FUNCTION_BLOCK SlaveAxisControl EXTENDS MasterAxisControl
VAR
	
	_PreviousAnglePosition		: LREAL;
	_PreviousLengthOfShaft		: LREAL;
	_PreviousWidthOfShaft		: LREAL;
	
	_xCoordPreviousRelative		: LREAL;
	_yCoordPreviousRelative		: LREAL;
	_xCoordPreviousGlobal		: LREAL;
	_yCoordPreviousGlobal		: LREAL;
	_xCoordGlobal				: LREAL;
	_yCoordGlobal				: LREAL;
	
	_SlaveOrderInChain			: LREAL;
	
END_VAR

METHOD CyclicUpdate : BOOL
VAR_INPUT
END_VAR
_Enable(Axis := _Axis);
_Reset(Axis := _Axis);
_ReadStatus(Axis := _Axis);
_MovePosAbs(Axis := _Axis);
_MovePosRel(Axis := _Axis);

_AnglePosition := _Axis.NcToPlc.ModuloActPos;

_xCoordRelative := _PreviousLengthOfShaft * COS(_PreviousAnglePosition * Pi / 180);
_yCoordRelative := _PreviousLengthOfShaft * SIN(_PreviousAnglePosition * Pi / 180);

_xCoordGlobal := _xCoordRelative + _xCoordPreviousGlobal;
_yCoordGlobal := _yCoordRelative + _yCoordPreviousGlobal;
END_METHOD

PROPERTY PreviousAnglePosition : LREAL
GET
PreviousAnglePosition := _PreviousAnglePosition;
END_GET
SET
_PreviousAnglePosition := PreviousAnglePosition;
END_SET
END_PROPERTY

PROPERTY PreviousLengthOfShaft : LREAL
GET
PreviousLengthOfShaft := _PreviousLengthOfShaft;
END_GET
SET
_PreviousLengthOfShaft := PreviousLengthOfShaft;
END_SET
END_PROPERTY

PROPERTY PreviousWidthOfShaft : LREAL
GET
PreviousWidthOfShaft := _PreviousWidthOfShaft;
END_GET
SET
_PreviousWidthOfShaft := PreviousWidthOfShaft;
END_SET
END_PROPERTY

PROPERTY PreviousXCoordGlobal : LREAL
GET
PreviousXCoordGlobal := _xCoordPreviousGlobal;
END_GET
SET
_xCoordPreviousGlobal := PreviousXCoordGlobal;
END_SET
END_PROPERTY

PROPERTY PreviousXCoordRelative : LREAL
GET
PreviousXCoordRelative := _xCoordPreviousRelative;
END_GET
SET
_xCoordPreviousRelative := PreviousXCoordRelative;
END_SET
END_PROPERTY

PROPERTY PreviousYCoordGlobal : LREAL
GET
PreviousYCoordGlobal := _yCoordPreviousGlobal;
END_GET
SET
_yCoordPreviousGlobal := PreviousYCoordGlobal;
END_SET
END_PROPERTY

PROPERTY PreviousYCoordRelative : LREAL
GET
PreviousYCoordRelative := _yCoordPreviousRelative;
END_GET
SET
_yCoordPreviousRelative := PreviousYCoordRelative;
END_SET
END_PROPERTY

PROPERTY SlaveOrderInChain : LREAL
GET
SlaveOrderInChain := _SlaveOrderInChain;
END_GET
SET
IF SlaveOrderInChain < 1 THEN
	_SlaveOrderInChain := 1;
ELSE
	_SlaveOrderInChain := SlaveOrderInChain;
END_IF
END_SET
END_PROPERTY

PROPERTY XCoordGlobal : LREAL
GET
XCoordGlobal := _xCoordGlobal;
END_GET
SET
END_SET
END_PROPERTY

PROPERTY YCoordGlobal : LREAL
GET
YCoordGlobal := _yCoordGlobal;
END_GET
SET
END_SET
END_PROPERTY

END_FUNCTION_BLOCK

(* stored: Version 1.1.0.1, ProductVersion 3.1.4024.12
   POU SlaveAxisControl: Id {d8ebd79d-dd1b-4835-8aa9-d1e613ab2927}, SpecialFunc None
   Folder Methods: Id {ba7939f0-e91b-4c7d-8597-9e28735743c9}
   Folder Properties: Id {145bc9ea-6d77-45cc-bdf2-55c818cf66d3}
   Method CyclicUpdate: Id {5135d1cb-d140-44b0-8571-d9917921e246}
   Property PreviousAnglePosition: Id {401de715-c68e-4c73-86c3-2ee5f70cc188}
   Get Get: Id {c24e600a-2903-48d6-b9fa-3eb40073854d}
   Set Set: Id {e69371f3-c7ba-4224-9e4f-7efc6379c7be}
   Property PreviousLengthOfShaft: Id {90993024-e3a5-40ea-a1bc-1dfa7608b3d9}
   Get Get: Id {a6ba4a2a-324e-4046-bbc4-71da89db077c}
   Set Set: Id {9257e878-1579-4f29-a04d-335e42f8fdb0}
   Property PreviousWidthOfShaft: Id {ed2c23fe-ac27-4767-a87c-98869ff059d0}
   Get Get: Id {0def12c1-0069-425d-a777-544b4142b55a}
   Set Set: Id {418a476b-a7db-49ae-ae56-37498f7e28d4}
   Property PreviousXCoordGlobal: Id {f382988b-a5c1-49a5-81c7-c8dd14a92cd5}
   Get Get: Id {f84f85ab-88e4-4e21-b24b-adb6624a1c56}
   Set Set: Id {0ef05fb8-dc4b-408c-86c5-4e4b91e6bc2a}
   Property PreviousXCoordRelative: Id {798c4aab-b7ef-457d-b724-f088d05a6dea}
   Get Get: Id {8d544cf3-aa74-48b7-9c12-82db2ee9f523}
   Set Set: Id {9d2e4602-1e87-42c2-9758-6b15640e0787}
   Property PreviousYCoordGlobal: Id {f30b318e-ad9b-4c68-8188-060d6aeb9081}
   Get Get: Id {09fc61f0-4634-4d40-8cc7-a259b3f7006d}
   Set Set: Id {e4ae6b0f-f3ae-4bf0-b5da-e73e86797cc8}
   Property PreviousYCoordRelative: Id {9f434607-08dc-4a17-b8ed-4e6ff10b48d0}
   Get Get: Id {bd34922a-db25-448f-9239-379c3b6ee94a}
   Set Set: Id {70254f2d-eb8f-4db5-9042-c2129c509e6d}
   Property SlaveOrderInChain: Id {d6fbf4e6-d766-4c80-b8a7-77b1098a9634}
   Get Get: Id {7379b388-49c4-4c50-aa05-8d7ed695ed24}
   Set Set: Id {eb16264c-02bc-406d-aaaa-9a3ad8cc66ba}
   Property XCoordGlobal: Id {7588ca51-1154-418a-a2f0-b31ed871ff04}
   Get Get: Id {afe87cc7-e156-4d7e-ab88-c1fb0a705f2b}
   Set Set: Id {c47d160f-9687-4d05-ad91-dd0a226d41ed}
   Property YCoordGlobal: Id {afdac74d-dfdb-4ec8-9d6b-986a5f4682b4}
   Get Get: Id {ac5da671-ff58-48ff-8745-f8581d93018e}
   Set Set: Id {c9c6c84f-a2b2-4210-9a2c-00d9e1bc7cff} *)
